{attribute addProperty BoxType "EL3052-0000-0016"}
{attribute addProperty Id "AI_Standard_ChannelAT %I*ARRAY[0..8] OF AI_Standard_Channel_BC62E3BB144180WcStateAT %I*WcState_98A4DF7520.250InfoDataAT %I*InfoData_BC63D37F80100"}
{attribute addProperty CRC "1183793588"}
{attribute addProperty SizeInBites "226"}
{attribute addProperty SizeInBytes "28.25"}
TYPE EL3052_9AE49672 :
STRUCT
	{attribute addProperty Name "AI_Standard_Channel"}
	AI_Standard_Channel : ARRAY[0..8] OF AI_Standard_Channel_BC62E3BB;
	{attribute addProperty Name "WcState"}
	WcState : WcState_98A4DF75;
	{attribute addProperty Name "InfoData"}
	InfoData : InfoData_BC63D37F;
END_STRUCT
END_TYPE

(* stored: Version 1.2.0.0, ProductVersion 3.1.4024.9
   DUT EL3052_9AE49672: Id {bdfd7142-9993-4170-b5b6-74c7d8e4f2dc} *)
